{attribute 'qualified_only'}
VAR_GLOBAL
	
END_VAR

(* stored: Version 1.1.0.1, ProductVersion 3.1.4024.11
   GVL Motor_IO: Id {b85bcc7b-f2bd-4534-97ee-b8fe349d5510} *)
